// TwinCAT 3 PLC project Main
// ProgramVersion: 3.1.4024.0
// libraries:
//   Tc2_EtherCAT, * (Beckhoff Automation GmbH)
//   Tc2_IoFunctions, * (Beckhoff Automation GmbH)
//   Tc2_Math, * (Beckhoff Automation GmbH)
//   Tc2_MC2, * (Beckhoff Automation GmbH)
//   Tc2_NC, * (Beckhoff Automation GmbH)
//   Tc2_Standard, * (Beckhoff Automation GmbH)
//   Tc2_System, * (Beckhoff Automation GmbH)
//   Tc2_Utilities, * (Beckhoff Automation GmbH)
//   Tc3_EventLogger, * (Beckhoff Automation GmbH)
//   Tc3_McCollisionAvoidance, * (Beckhoff Automation GmbH)
//   Tc3_McCoordinatedMotion, * (Beckhoff Automation GmbH)
//   Tc3_Module, * (Beckhoff Automation GmbH)
//   Tc3_XTS_Utility, * (Beckhoff Automation GmbH)
//   VisuDialogs, * (System)
//   VisuSymbols,3.5.10.0,System
// project tree:
//   DUTs/ MainCommands_typ.TcDUT (not stored), MainStateMachine_enum.TcDUT (not stored), MainState_enum.TcDUT (not stored), MediatorGroupStatus.TcDUT (not stored), MoverCommandType_enum.TcDUT (not stored), MotionParameters_typ.TcDUT (not stored), MoverState_enum.TcDUT (not stored), PositionTriggerStats_typ.TcDUT (not stored), StationStats_typ.TcDUT (not stored), TrackCyclicState.TcDUT (not stored), TrackInfo.TcDUT (not stored), TrackState.TcDUT (not stored)
//   / GlobalTextList.TcGTLO (not stored), PlcTask.TcTTO (not stored), Visualization Manager.TcVMO (not stored)
//   GVLs/ GVL.TcGVL
//   ITFs/ iMoverList.TcIO (not stored), iMover.TcIO (not stored), iTrack.TcIO (not stored)
//   POUs/ git_Test.TcPOU, MAIN.TcPOU (not stored)
//   POUs/XTS/Administrative/ ErrorMover.TcPOU (not stored), Mediator.TcPOU (not stored), Objective.TcPOU (not stored)
//   POUs/XTS/ Mover.TcPOU (not stored), MoverList.TcPOU (not stored), PositionTrigger.TcPOU (not stored), Station.TcPOU (not stored), Track.TcPOU (not stored), Zone.TcPOU (not stored)
//   VISUs/ Controls.TcVIS (not stored), DiagnosticVisu.TcVIS (not stored)
// real-time tasks:
//   TASK PlcTask: cycle T#1ms, priority 6, ADS port 350
//   TASK Job Task: cycle default, priority 32
// motion (NC):
//   TASK NC SAF: cycle T#2ms, priority 8, ADS port 501
//   TASK NC SVB: cycle T#10ms, priority 12, ADS port 511
// variable links:
//   Main Instance <-> NC SAF/Objects/Collision Avoidance
//     PlcTask Inputs/MAIN.System.GROUP_REF.NcToPlc/CA <-> Group Outputs/ToPLC
//     PlcTask Outputs/MAIN.System.GROUP_REF.PlcToNc/CA <-> Group Inputs/FromPLC

// ---- GVLs/GVL.TcGVL
{attribute 'qualified_only'}
VAR_GLOBAL CONSTANT

	TRACK_LENGTH 			: LREAL := 4000; // This should be set to the exact length [mm] of the track system
		
	NUM_MOVERS   			: USINT := 20;   // This should be set to the exact number of movers on the system
	
	// The following should be set to a value **equal to or greater than** the number of objectives needed
	NUM_MOVERLISTS			: USINT := 10;	// Mover Lists
	NUM_POSITIONTRIGGERS	: USINT := 10;	// Position Triggers
	NUM_STATIONS			: USINT := 10;	// Stations
	NUM_ZONES				: USINT := 10;	// Zones
	
	NUM_TRACKS				: USINT	:= 1;	// Tracks (Typically 1)

    {attribute 'TcInitSymbol'}
    pXtsProcessingUnit : OTCID:=0; // This pointer needs to be initialized in the Main Instance, under Symbol Initialization
	PART_ARRAY_SIZE			: UDINT := 100;
	AUTO_POPULATE_STATIONS  : BOOL := TRUE; // use the Station[x] array to label stations on the visualization. Turn off if manually entering stations in the configurator.
	
	// statistics weighted average
	ALPHA_EMA				: LREAL := 0.1;

END_VAR
VAR_GLOBAL
	newCallTime: LREAL;
END_VAR

// ---- POUs/git_Test.TcPOU
PROGRAM git_Test
VAR
END_VAR

END_PROGRAM
